PROGRAM MAIN
VAR
END_VAR

END_PROGRAM

(* stored: Version 1.1.0.1
   POU MAIN: Id {637ad8fb-d548-4a62-8ad9-cf235c97c63c} *)
